// Mitsubishi GX Works2 project: BookEX2_1 CrossRoad   PLC: Q13UDV

// global labels: CrossRoad
VAR_GLOBAL
  bStartNorth AT M0 : BOOL;
  bStartEast AT M1 : BOOL;
  bStartSouth AT M2 : BOOL;
  bStartWest AT M3 : BOOL;
  bMode AT M4 : BOOL;
  bNorthR AT Y0 : BOOL;
  bNorthY AT Y1 : BOOL;
  bNorthA AT Y2 : BOOL;
  bNorthG AT Y3 : BOOL;
  bEastR AT Y4 : BOOL;
  bEastY AT Y5 : BOOL;
  bEastA AT Y6 : BOOL;
  bEastG AT Y7 : BOOL;
  bSouthR AT Y8 : BOOL;
  bSouthY AT Y9 : BOOL;
  bSouthA AT Y0A : BOOL;
  bSouthG AT Y0B : BOOL;
  bWestR AT Y0C : BOOL;
  bWestY AT Y0D : BOOL;
  bWestA AT Y0E : BOOL;
  bWestG AT Y0F : BOOL;
  iTimeNorth AT D10 : INT;
  iTimeEast AT D11 : INT;
  iTimeSouth AT D12 : INT;
  iTimeWest AT D13 : INT;
  iLampNorth AT D20 : INT;
  iLampEast AT D21 : INT;
  iLampSouth AT D22 : INT;
  iLampWest AT D23 : INT;
  bActNorth AT M10 : BOOL;
  bActEast AT M11 : BOOL;
  bActSouth AT M12 : BOOL;
  bActWest AT M13 : BOOL;
  bStopNorth AT M20 : BOOL;
  bStopEast AT M21 : BOOL;
  bStopSouth AT M22 : BOOL;
  bStopWest AT M23 : BOOL;
  bTimerOffNorth AT M30 : BOOL;
  bTimerOfftEast AT M31 : BOOL;
  bTimeOffSouth AT M32 : BOOL;
  bTimeOffWest AT M33 : BOOL;
END_VAR
VAR_GLOBAL CONSTANT
  ctOnTimeG : TIME := T#15s;
  ciDigitBlink : INT := 10;
END_VAR
// user libraries (not included): HMI

FUNCTION_BLOCK LoopCtrl
VAR_INPUT
  b_Mode : BOOL;
  b_Stop1 : BOOL;
END_VAR
VAR_OUTPUT
  b_Start1 : BOOL;
END_VAR
VAR_INPUT
  b_Stop2 : BOOL;
  b_Stop3 : BOOL;
  b_Stop4 : BOOL;
END_VAR
VAR_OUTPUT
  b_Start2 : BOOL;
  b_Start3 : BOOL;
  b_Start4 : BOOL;
END_VAR
VAR
  Phase : INT;
END_VAR
VAR_INPUT
  b_Act1 : BOOL;
  b_Act2 : BOOL;
  b_Act3 : BOOL;
  b_Act4 : BOOL;
END_VAR
;
IF NOT b_Mode THEN
	b_Start1 := FALSE;
	b_Start2 := FALSE;
	b_Start3 := FALSE;
	b_Start4 := FALSE;
	Phase := 0;
	RETURN;
END_IF;

CASE Phase MOD 8 OF
	0 : (* Top *)
			b_Start1 := TRUE;
			b_Start2 := FALSE;
			b_Start3 := FALSE;
			b_Start4 := FALSE;
			IF b_Act1 THEN
				Phase := Phase + 1;
			END_IF;
	1 : IF b_Stop1 THEN
				Phase := Phase + 1;
			END_IF;			
	2 : (* Right *)
			b_Start1 := FALSE;
			b_Start2 := TRUE;
			b_Start3 := FALSE;
			b_Start4 := FALSE;
			IF b_Act2 THEN
				Phase := Phase + 1;
			END_IF;
	3 : IF b_Stop2 THEN
				Phase := Phase + 1;
			END_IF;			
	4 : (* Bottom *)
			b_Start1 := FALSE;
			b_Start2 := FALSE;
			b_Start3 := TRUE;
			b_Start4 := FALSE;
			IF b_Act3 THEN
				Phase := Phase + 1;
			END_IF;
	5 : IF b_Stop3 THEN
				Phase := Phase + 1;
			END_IF;			
	6 : (* Left *)
			b_Start1 := FALSE;
			b_Start2 := FALSE;
			b_Start3 := FALSE;
			b_Start4 := TRUE;
			IF b_Act4 THEN
				Phase := Phase + 1;
			END_IF;
	7 : IF b_Stop4 THEN
				Phase := 0;
			END_IF;			
END_CASE;
END_FUNCTION_BLOCK

FUNCTION_BLOCK TrafficLamp
VAR_INPUT
  b_Start : BOOL;
END_VAR
VAR_OUTPUT
  b_Act : BOOL;
  b_Stop : BOOL;
  i_Cnt : INT;
END_VAR
VAR
  Phase : INT;
  fbTimer1 : TON;
  fbTimer2 : TON;
END_VAR
VAR_INPUT
  t_TimeG : TIME;
END_VAR
VAR_OUTPUT
  b_G : BOOL;
  b_Y : BOOL;
  b_R : BOOL;
END_VAR
VAR_INPUT
  b_Mode : BOOL;
END_VAR
;
IF NOT b_Start THEN
	IF b_Mode THEN
		b_G := FALSE;
		b_Y := FALSE;
		b_R := TRUE;
	ELSE
		b_G := FALSE;
		b_Y := SM412;
		b_R := FALSE;	
	END_IF;
	b_Act := FALSE;
	b_Stop := FALSE;
	i_Cnt := 0;
	Phase := 0;
	fbTimer1(IN:=FALSE);
	fbTimer2(IN:=FALSE);
	RETURN;
END_IF;
 
CASE Phase OF
	0 : (* Start *)
			b_G := FALSE;
			b_Y := FALSE;
			b_R := FALSE;
			b_Act := TRUE;
			b_Stop := FALSE;
			Phase := 1;
	1 : (* Green *)
			b_G := TRUE;
			fbTimer1(IN := TRUE, PT:=t_TimeG);	
			IF fbTimer1.Q THEN
				fbTimer1(IN:=FALSE);
				b_G := FALSE;
				Phase := 2;
			END_IF;
	2 : (* Yellow *)
			b_Y := TRUE;
			fbTimer2(IN := TRUE, PT:=T#3s);	
			IF fbTimer2.Q THEN
				fbTimer2(IN:=FALSE);
				b_Y := FALSE;
				Phase := 3;
			END_IF;
	3 : (* Red *)
			b_R := TRUE;
			b_Stop := TRUE;
			b_Act := FALSE;
END_CASE;

IF b_G THEN
	i_Cnt := TIME_TO_INT(DIV_TIME(t_TimeG, 500) - DIV_TIME(fbTimer1.ET, 500));
ELSE
	i_Cnt := 0;
END_IF;
END_FUNCTION_BLOCK

FUNCTION_BLOCK WalkLamp
VAR_INPUT
  i_Cnt : INT;
END_VAR
VAR_OUTPUT
  i_Time : INT;
  i_Lamp : INT;
  b_OffFlag : BOOL;
END_VAR
VAR
  ix : INT;
  iy : INT;
END_VAR
VAR_INPUT
  i_Blink : INT;
END_VAR
;
IF i_Cnt = 0 THEN
	i_Time := 0;
	i_Lamp := 1;
	b_OffFlag := TRUE;
ELSE
	ix := i_Cnt / 2;	iy := i_Cnt MOD 2;
	i_Time := ix;
	IF i_Cnt < 2 THEN b_OffFlag := TRUE; ELSE  b_OffFlag := FALSE; END_IF;
	IF ix > i_Blink THEN
		i_Lamp := 2;
	ELSE
		IF iy = 1 THEN
			i_Lamp := 2;
		ELSE
			i_Lamp := 0;
		END_IF;
	END_IF;
END_IF;
END_FUNCTION_BLOCK

PROGRAM Cross
VAR
  TrafficLamp_1 : TrafficLamp;
  WalkLamp_1 : WalkLamp;
  TrafficLamp_2 : TrafficLamp;
  TrafficLamp_3 : TrafficLamp;
  TrafficLamp_4 : TrafficLamp;
  WalkLamp_2 : WalkLamp;
  WalkLamp_3 : WalkLamp;
  WalkLamp_4 : WalkLamp;
  LoopCtrl_1 : LoopCtrl;
  iCnt2 : INT;
  TrafficLamp_5 : TrafficLamp;
END_VAR
(* structured ladder/FBD written out as ST: instructions are called as NAME(EN, inputs, outputs); _pN, _eN, _tN stand for wires *)
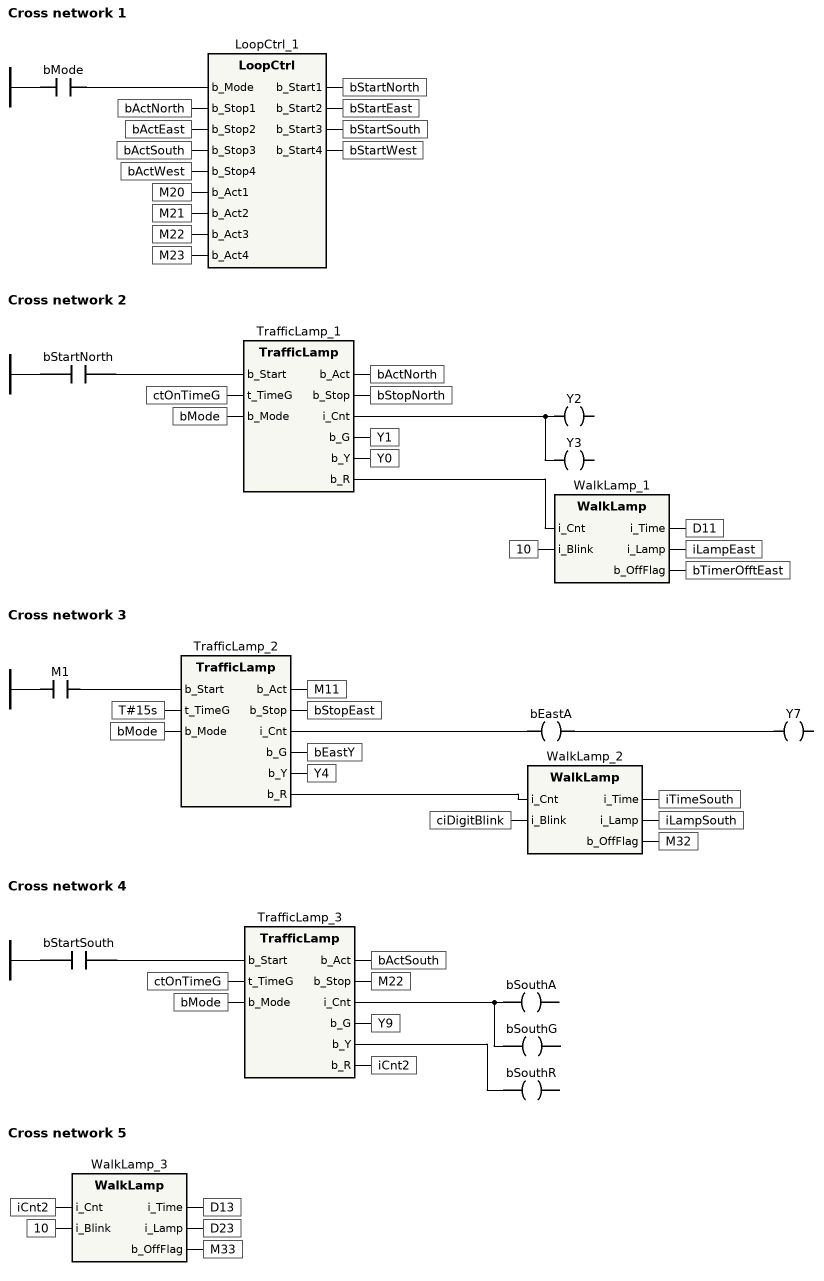
(* network 1 *)
LoopCtrl_1(b_Mode := bMode, b_Stop1 := bActNorth, b_Stop2 := bActEast, b_Stop3 := bActSouth, b_Stop4 := bActWest, b_Act1 := M20, b_Act2 := M21, b_Act3 := M22, b_Act4 := M23, b_Start1 => bStartNorth, b_Start2 => bStartEast, b_Start3 => bStartSouth, b_Start4 => bStartWest);
(* network 2 *)
TrafficLamp_1(b_Start := bStartNorth, t_TimeG := ctOnTimeG, b_Mode := bMode, b_Act => bActNorth, b_Stop => bStopNorth, b_G => Y1, b_Y => Y0);
Y2 := TrafficLamp_1.i_Cnt;
Y3 := TrafficLamp_1.i_Cnt;
WalkLamp_1(i_Cnt := TrafficLamp_1.b_R, i_Blink := 10, i_Time => D11, i_Lamp => iLampEast, b_OffFlag => bTimerOfftEast);
(* network 3 *)
TrafficLamp_2(b_Start := M1, t_TimeG := T#15s, b_Mode := bMode, b_Act => M11, b_Stop => bStopEast, b_G => bEastY, b_Y => Y4);
bEastA := TrafficLamp_2.i_Cnt;
Y7 := TrafficLamp_2.i_Cnt;
WalkLamp_2(i_Cnt := TrafficLamp_2.b_R, i_Blink := ciDigitBlink, i_Time => iTimeSouth, i_Lamp => iLampSouth, b_OffFlag => M32);
(* network 4 *)
TrafficLamp_3(b_Start := bStartSouth, t_TimeG := ctOnTimeG, b_Mode := bMode, b_Act => bActSouth, b_Stop => M22, b_G => Y9, b_R => iCnt2);
bSouthA := TrafficLamp_3.i_Cnt;
bSouthG := TrafficLamp_3.i_Cnt;
bSouthR := TrafficLamp_3.b_Y;
(* network 5 *)
WalkLamp_3(i_Cnt := iCnt2, i_Blink := 10, i_Time => D13, i_Lamp => D23, b_OffFlag => M33);
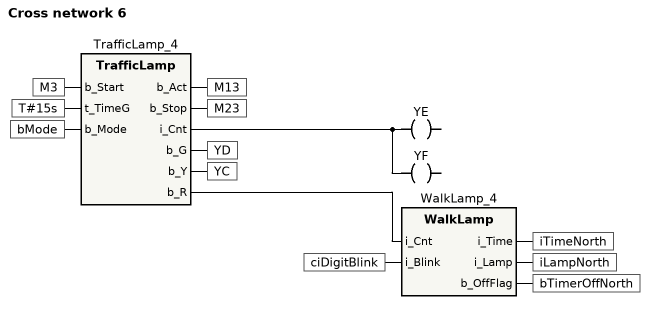
(* network 6 *)
TrafficLamp_4(b_Start := M3, t_TimeG := T#15s, b_Mode := bMode, b_Act => M13, b_Stop => M23, b_G => YD, b_Y => YC);
YE := TrafficLamp_4.i_Cnt;
YF := TrafficLamp_4.i_Cnt;
WalkLamp_4(i_Cnt := TrafficLamp_4.b_R, i_Blink := ciDigitBlink, i_Time => iTimeNorth, i_Lamp => iLampNorth, b_OffFlag => bTimerOffNorth);
END_PROGRAM
